FUNCTION_BLOCK FB_GetTimePML
VAR_INPUT
END_VAR
VAR_OUTPUT
	PML_Time		: ARRAY [0..6] OF DINT;
END_VAR
VAR
	fbGetTime		: NT_GetTime;
	tonInterval		: TON;
	tInterval		: TIME := T#100ms;
END_VAR


tonInterval(	IN := NOT tonInterval.Q,
				PT := tInterval,
				Q =>,
				ET =>	);

fbGetTime(	NETID:= '', 
			START:= tonInterval.Q, 
			TMOUT:= T#5S, 
			BUSY=> , 
			ERR=> , 
			ERRID=> , 
			TIMESTR=> 	);


PML_Time := TIMESTRUCT_TO_PackMLTime(fbGetTime.TIMESTR);

END_FUNCTION_BLOCK

(* stored: Version 1.1.0.1, ProductVersion 3.1.4024.2
   POU FB_GetTimePML: Id {022b1905-7544-44a7-8454-cc0c49374b80}, SpecialFunc None *)
